Universal Robots PolyScope program: reciprocal_p3_2.urp

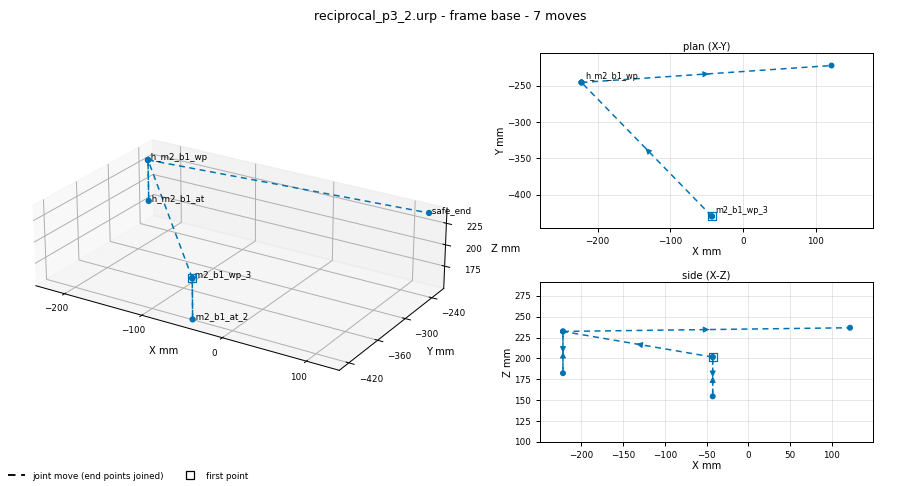
[picture p0: tool path of reciprocal_p3_2.urp in frame base, 7 of 7 moves have a stored position in this frame; points joined in program order, loops and branches not executed]
Program reciprocal_p3_2 (installation=default directory=/programs/ITER createdIn=5.3.1.64192 lastSavedIn=5.3.1.64192 robotSerialNumber=20195300365)
Calibrated DH parameters: a=[-0.000093, -0.190649, -0.212673, 0.000091, -0.000205, 0]; d=[0.151591, 44.061648, -42.488068, -1.442789, 0.085322, 0.091911]; alpha=[1.570082, -0.003447, 0.007513, 1.572293, -1.571904, 0]; deltaTheta=[0, -0.672656, 0.728185, -0.055522, 0.000005, 0]
Robot Program (runOnlyOnce=true)
  URCap Gripper Activate (Robotiq_Grippers, Robotiq Inc.) dataModel(ResetAndActivateKey=false)
  URCap Gripper (Robotiq_Grippers, Robotiq Inc.) dataModel(position=50.0, force=100.0, speed=100.0, positionInDouble=50.0, forceInDouble=100.0, speedInDouble=100.0, slaveIds=[9], blocking=true)
  Folder Mid_2
    MoveJ speed 60 deg/s, acceleration 80 deg/s^2 (useActiveTCP=true) feature=Base
      Waypoint m2_b1_wp_3: TCP in base x=-42.705 y=-429.628 z=201.674 mm, rx=2.2154 ry=2.1777 rz=0.0173 rad; joints [-78.53, -120.549, -78.862, -69.183, 91.892, -257.242] deg
      Waypoint m2_b1_at_2: TCP in base x=-42.72 y=-429.623 z=154.534 mm, rx=2.2155 ry=2.1777 rz=0.0173 rad; joints [-78.548, -125.214, -84.966, -58.413, 91.858, -257.198] deg
      URCap Gripper (Robotiq_Grippers, Robotiq Inc.) dataModel(position=100.0, force=100.0, speed=100.0, positionInDouble=100.0, forceInDouble=100.0, speedInDouble=100.0, slaveIds=[9], blocking=true)
      Waypoint m2_b1_wp_4: TCP in base x=-42.705 y=-429.628 z=201.674 mm, rx=2.2154 ry=2.1777 rz=0.0173 rad; joints [-78.53, -120.549, -78.862, -69.183, 91.892, -257.242] deg
      Waypoint h_m2_b1_wp: TCP in base x=-222.193 y=-245.34 z=232.403 mm, rx=-3.1314 ry=0.0205 rz=0.0123 rad; joints [-108.936, -94.247, -105.13, -70.966, 89.712, -197.837] deg
      Waypoint h_m2_b1_at: TCP in base x=-222.194 y=-245.343 z=182.32 mm, rx=-3.1314 ry=0.0205 rz=0.0122 rad; joints [-108.96, -99.771, -113.792, -56.782, 89.658, -197.776] deg
      URCap Gripper (Robotiq_Grippers, Robotiq Inc.) dataModel(position=50.0, force=100.0, speed=100.0, positionInDouble=50.0, forceInDouble=100.0, speedInDouble=100.0, slaveIds=[9], blocking=true)
      Waypoint h_m2_b1_wp: TCP in base x=-222.193 y=-245.34 z=232.403 mm, rx=-3.1314 ry=0.0205 rz=0.0123 rad; joints [-108.936, -94.247, -105.13, -70.966, 89.712, -197.837] deg
  MoveJ speed 60 deg/s, acceleration 80 deg/s^2 (useActiveTCP=true) feature=Base
    Waypoint safe_end: TCP in base x=121.882 y=-222.057 z=236.793 mm, rx=2.2146 ry=2.209 rz=-0.0386 rad; joints [-29.832, -71.908, -123.399, -74.268, 88.825, -209.331] deg
